Fanuc KAREL source: kt00160.compact.KL

PROGRAM KT00160
%STACKSIZE=65535
%PRIORITY=65535
%NOLOCKGROUP
VAR
H1 : ARRAY[2] OF SHORT
H2 : ARRAY[2] OF SHORT
OUT : REAL
BEGIN
H1[1]=2
H2[1]=3
H1[1]=2
H2[1]=3
OUT=((H1[1] DIV H2[1]))
END KT00160
